TYPE Array8_LReal :
UNION
	arrByte			:ARRAY[0..7] OF BYTE;
	rValue			:LREAL;
END_UNION
END_TYPE

(* stored: Version 1.1.0.1
   DUT Array8_LReal: Id {a242b221-9eac-4b96-9a07-24d05cc8ad50} *)
